{attribute 'conditionalshow_all_locals'}
{attribute 'no_explicit_call' := 'JsonDecoder is a class, do not call'}
FUNCTION_BLOCK JsonDecoder
VAR
  _key : STRING;
  _jsonPtr : POINTER TO BYTE;
  _memPtr : POINTER TO BYTE;
  
  _elements : ARRAY[0..ParameterList.MaxJsonAssignments] OF JsonElement;
  _elementCount : UINT;  
  
  _root : JsonNode;
  _nodes : ARRAY[0..ParameterList.MaxJsonAssignments] OF JsonNode;
  _nodeCount : UINT;
  
  _el : JsonElementType;
END_VAR
VAR_OUTPUT
  Error : BOOL;
  ErrorMessage : STRING;
END_VAR

METHOD PROTECTED _Element : IJsonElement
VAR_INPUT
  node : POINTER TO JsonNode;
  readPtr : POINTER TO BYTE;
END_VAR
VAR
  writePtr : POINTER TO BYTE;
  child : POINTER TO JsonNode;
END_VAR
// get next key, for part1.part2.part3, part1 is yieled
writePtr := ADR(_key);
WHILE readPtr^ <> 16#0 AND_THEN readPtr^ <> 16#2E AND_THEN readPtr^ <> 16#5B AND_THEN readPtr^ <> 16#5D // eof, . or [
DO
  writePtr^ := readPtr^;
  writePtr := writePtr + 1;
  readPtr := readPtr + 1;
END_WHILE
writePtr^ := 0;

IF readPtr^ <> 0 AND_THEN readPtr^ = 16#5D  // skip ]
THEN 
  readPtr := readPtr + 1; 
END_IF

IF readPtr^ <> 0 AND_THEN readPtr^ = 16#2E // skip .  
THEN 
  readPtr := readPtr + 1;
END_IF  

IF readPtr^ <> 0 AND_THEN readPtr^ = 16#5B  // skip [  
THEN 
  readPtr := readPtr + 1;  
END_IF 

// search for child with current key, if a match is found
// check if we are at the end of the path and return the potential value,
// otherwise recurse to next level
child := node^.FirstChild;
WHILE child <= node^.LastChild
DO
  IF child^.Name = _key
  THEN
    IF child^.FirstChild <> 0 AND_THEN child^.FirstChild^.IsArray // we are dealing with an array
    THEN
      _Element := THIS^._Element(child^.FirstChild, readPtr);
    ELSIF readPtr^ <> 0
    THEN
      _Element := THIS^._Element(child, readPtr);    
    ELSIF NOT child^.IsArray AND_THEN child^.Element <> 0 // direct access, exact match
    THEN
      _Element := child^.Element^;
    END_IF
	END_IF
  
  IF _Element <> 0
  THEN
    RETURN;
	END_IF
  child := child^.Next;
END_WHILE
END_METHOD

METHOD PROTECTED Abort
VAR_IN_OUT CONSTANT
  errorMessage : STRING;
END_VAR
THIS^.ErrorMessage := errorMessage;
THIS^.Error := TRUE;
END_METHOD

METHOD PROTECTED AddElement
VAR_INPUT
  node : POINTER TO JsonNode;
END_VAR
VAR
  element : POINTER TO JsonElement;
END_VAR
element := ADR(_elements) + SIZEOF(JsonElement) * _elementCount;
element^.ValueType := _el;
element^.StartPtr := _memPtr;
element^.EndPtr := _jsonPtr;
_elementCount := _elementCount + 1;

node^.Element := element;
END_METHOD

METHOD PROTECTED AddNode : POINTER TO JsonNode
VAR_INPUT
  node : POINTER TO JsonNode;
END_VAR
VAR
  namePtr : POINTER TO BYTE;
  memPtr : POINTER TO BYTE;
END_VAR
AddNode := ADR(_nodes) + SIZEOF(JsonNode) * _nodeCount;
IF node^.LastChild <> 0
THEN
  node^.LastChild^.Next := AddNode;
  node^.LastChild := AddNode;
ELSE
  node^.FirstChild := AddNode;
  node^.LastChild := AddNode;
END_IF

// set node name
namePtr := ADR(AddNode^.Name);
memPtr := _memPtr;
WHILE memPtr <> _jsonPtr
DO
  namePtr^ := memPtr^;
  namePtr := namePtr + 1;
  memPtr := memPtr + 1;
END_WHILE
namePtr^ := 0;
// reset elements
AddNode^.IsArray := FALSE;
AddNode^.FirstChild := 0;
AddNode^.LastChild := 0;
_nodeCount := _nodeCount + 1;
END_METHOD

METHOD Decode
VAR_IN_OUT CONSTANT
  json : STRING;
END_VAR
_jsonPtr := ADR(json);
_elementCount := 0;
_nodeCount := 0;

Error := FALSE;

WHILE _jsonPtr^ <> 0
DO
  SkipWhitespaces();

  _el := GuessElementType();
  IF _el = JsonElementType.Object
  THEN 
    ParseObject(ADR(_root));
  ELSIF _el = JsonElementType.Arry
  THEN
    _memPtr := _jsonPtr;
    _root.FirstChild := AddNode(ADR(_root));
    _root.FirstChild^.Name := 'array';
    ParseArray(_root.FirstChild);
  ELSE
    Abort('Unexpected character');    
  END_IF  
  
  _jsonPtr := _jsonPtr + 1;
END_WHILE
END_METHOD

METHOD Element : IJsonElement
VAR_IN_OUT CONSTANT
  path : STRING;
END_VAR
Element := _Element(ADR(_root), ADR(path));
END_METHOD

METHOD PROTECTED GuessElementType : JsonElementType
VAR_INPUT
END_VAR
CASE _jsonPtr^
OF
  16#22: // "
    GuessElementType := JsonElementType.Strng;
  16#30..16#39, // 0-9
  16#2B, // +
  16#2D, // -
  16#2E, // .
  16#65, // e
  16#45: // E
    GuessElementType := JsonElementType.Number;    
  16#7B: // {
    GuessElementType := JsonElementType.Object;
  16#5B: // [
    GuessElementType := JsonElementType.Arry;
  16#66, // f
  16#74: // t
    GuessElementType := JsonElementType.Boolean;
  16#6E: // n
    GuessElementType := JsonElementType.Null;      
END_CASE
END_METHOD

METHOD PROTECTED IntToString
VAR_INPUT
  element : INT;
END_VAR
VAR_IN_OUT CONSTANT
  str : STRING;
END_VAR
VAR
  writePtr : POINTER TO BYTE;
  reversePtr : POINTER TO BYTE;  
  endPtr : POINTER TO BYTE;  
END_VAR
writePtr := ADR(str);
reversePtr := ADR(str);

// we have to write the index in reverse, for element 12, we first build a string
// that looks like 21 and then we reverse it
// todo: test if a seperate branch for element < 10 is faster than doing the generic algorithm for this edge case as well
REPEAT
  writePtr^ := INT_TO_BYTE(element MOD 10) + 16#30; writePtr := writePtr + 1;
  element := element / 10; 
UNTIL element = 0 END_REPEAT
writePtr^ := 0;

// reverse string with XOR swap algorithm
endPtr := writePtr - 1;
WHILE reversePtr < endPtr
DO
  // swap first and last
  reversePtr^ := endPtr^ XOR reversePtr^;
  endPtr^ := reversePtr^ XOR endPtr^;
  reversePtr^ := endPtr^ XOR reversePtr^;
  
  reversePtr := reversePtr + 1;
  endPtr := endPtr - 1;
END_WHILE
END_METHOD

METHOD PROTECTED ParseArray
VAR_INPUT
  node : POINTER TO JsonNode;
END_VAR
VAR
  child : POINTER TO JsonNode;
  elements : INT;
END_VAR
node^.IsArray := TRUE;
_jsonPtr := _jsonPtr + 1;

REPEAT

  _memPtr := _jsonPtr; // we set the name by index later on
  child := AddNode(node);
  IntToString(elements, child^.Name);
  elements := elements + 1;
  ParseElement(child);
  
  // got another element in this object?
  IF _jsonPtr^ = 16#2C // ,
  THEN
    _jsonPtr := _jsonPtr + 1; // ,
    SkipWhitespaces();      
  END_IF    

UNTIL _jsonPtr^ = 16#5D OR_ELSE _jsonPtr^ = 0 END_REPEAT // } or EOF

IF _jsonPtr^ <> 0
THEN
  // skip ]
  _jsonPtr := _jsonPtr + 1;
END_IF
END_METHOD

METHOD PROTECTED ParseElement
VAR_INPUT
  node : POINTER TO JsonNode;  
END_VAR
VAR
  child : POINTER TO JsonNode;
END_VAR
SkipWhitespaces();
_el := GuessElementType();
CASE _el
OF
  JsonElementType.Strng:
    // skip " and additional whitespaces
    _jsonPtr := _jsonPtr + 1;
    _memPtr := _jsonPtr;
    SkipString();
    AddElement(node);
    // skip "
    _jsonPtr := _jsonPtr + 1;    
  
  JsonElementType.Number:
    _memPtr := _jsonPtr;
    SkipNumber();
    AddElement(node);
    
  JsonElementType.Object:
    // add . to the key and continue with the next object
    //_pathPtr^ := 16#2E;
    //_pathPtr := _pathPtr + 1;
    ParseObject(node);
  
    // remove . from the key
    //_pathPtr^ := 0;
    //_pathPtr := _pathPtr - 1;
  
  JsonElementType.Arry:
  
    child := AddNode(node);
    child^.Name := '';
    ParseArray(child);
    
  JsonElementType.Boolean:
    _memPtr := _jsonPtr;
    SkipBoolean();
    AddElement(node);
    
  JsonElementType.Null:
    _memPtr := _jsonPtr;
    _jsonPtr := _jsonPtr + 4; // null
    AddElement(node);
ELSE
  Abort('Unexpected character');
  RETURN;
END_CASE

SkipWhitespaces();
END_METHOD

METHOD PROTECTED ParseObject
VAR_INPUT
  node : POINTER TO JsonNode;  
END_VAR
VAR
  child : POINTER TO JsonNode;
  childNamePtr : POINTER TO BYTE;
END_VAR
// skip {
_jsonPtr := _jsonPtr + 1;
SkipWhitespaces();

REPEAT

  _el := GuessElementType();
  IF _el <> JsonElementType.Strng
  THEN
    Abort('Unexpected character');
    RETURN;    
  END_IF
  
  // skip "
  _jsonPtr := _jsonPtr + 1;
  _memPtr := _jsonPtr;
  SkipString();
  
  // chain key
  child := AddNode(node);
    
  // skip " and additional whitespaces
  _jsonPtr := _jsonPtr + 1;
  SkipWhitespaces();
  
  IF _jsonPtr^ <> 16#3A // :
  THEN
    Abort('Expected colon');
    RETURN;
  END_IF
  
  // skip :
  _jsonPtr := _jsonPtr + 1;
  ParseElement(child);
  
  // got another element in this object?
  IF _jsonPtr^ = 16#2C // ,
  THEN
    _jsonPtr := _jsonPtr + 1; // ,
    SkipWhitespaces();      
  END_IF  
  
UNTIL _jsonPtr^ = 16#7D OR_ELSE _jsonPtr^ = 0 END_REPEAT // } or EOF

IF _jsonPtr^ <> 0
THEN
  // skip }
  _jsonPtr := _jsonPtr + 1;
END_IF
END_METHOD

METHOD PROTECTED SkipBoolean
_jsonPtr := _jsonPtr + 4; // true

IF _jsonPtr^ = 16#66 // f
THEN
  _jsonPtr := _jsonPtr + 1; // false
END_IF
END_METHOD

METHOD PROTECTED SkipNumber
VAR
  ch : BYTE;
END_VAR
ch := _jsonPtr^;
WHILE (ch >= 16#30 AND_THEN ch <= 16#39) OR_ELSE ch = 16#2B OR_ELSE ch = 16#2D OR_ELSE ch = 16#2E OR_ELSE ch = 16#65 OR_ELSE ch = 16#45
DO
  _jsonPtr := _jsonPtr + 1;
  ch := _jsonPtr^;
END_WHILE
END_METHOD

METHOD PROTECTED SkipString
WHILE _jsonPtr^ <> 16#22
DO
  _jsonPtr := _jsonPtr + 1;
END_WHILE
END_METHOD

METHOD PROTECTED SkipWhitespaces
VAR
  ch : BYTE;
END_VAR
ch := _jsonPtr^;
WHILE ch > 0 AND_THEN ch <= 16#20
DO
  _jsonPtr := _jsonPtr + 1;
  ch := _jsonPtr^;
END_WHILE
END_METHOD

END_FUNCTION_BLOCK

(* stored: Version 1.1.0.1, ProductVersion 3.1.4024.12
   POU JsonDecoder: Id {c2bd40df-6169-4fb7-bccc-6fe5055a7ea3}, SpecialFunc None
   Method _Element: Id {01b90b91-98df-458d-95e0-7ae03947dbdb}
   Method Abort: Id {151abc50-572e-41de-9235-590a6cc2cb06}
   Method AddElement: Id {b4920f3e-12a7-4d6b-b494-42db676d6673}
   Method AddNode: Id {489314ba-53d4-43bd-a926-ca72da578204}
   Method Decode: Id {9e0a559b-3090-4700-8907-be0f1642151e}
   Method Element: Id {4a76f022-7ad8-455a-86cd-e4ff5a774583}
   Method GuessElementType: Id {34940981-ada5-4521-bbcd-34f0ecb406f1}
   Method IntToString: Id {0844489d-f692-4848-a8a9-c7fd5ee901c8}
   Method ParseArray: Id {31f9e53c-038a-44b5-a16c-e5766a0048e5}
   Method ParseElement: Id {78f23aa0-bb02-4013-930a-f14a7bc442cb}
   Method ParseObject: Id {d3f57aad-1f9b-4dd9-890f-af9c01be5099}
   Method SkipBoolean: Id {8891d801-d872-42b4-a283-4d50aacd8df8}
   Method SkipNumber: Id {77969f1c-9894-42e4-81b6-8fc4acc31c50}
   Method SkipString: Id {1acc1bd3-5568-4718-af78-edb71be6e7a9}
   Method SkipWhitespaces: Id {eb42f950-84b2-4370-a0c4-aff9ce5ce2f4} *)
